// Brief: Master Arm Master Slave Control
FUNCTION_BLOCK PUBLIC FB_StateCtrlInit EXTENDS FB_MasterArmCtrlBase
VAR_INPUT
END_VAR
VAR_OUTPUT
END_VAR
VAR
	m_jnt7SelfCheckVel : LREAL :=180*g_deg2Rad;
	m_jnt7HalfMotionRange : LREAL := 1.75*PI+0.26;
	m_jnt7LimitErr :LREAL := 5*g_deg2Rad;
	m_jnt7CenterPos :LREAL;
	// 0: driver on; 1: joint 7 move to upper limit, 2: joint 7 mvoe to center
	m_initState :INT :=0;
END_VAR

// override this function in each exact controller
METHOD PROTECTED calcCmdJntPos : BOOL

VAR_IN_OUT CONSTANT
	i_slaveIdx :INT;
	i_shoulderPose :ST_Frame;
	i_masterArm :FB_MasterArm;
	i_slaveStatus :ST_SlaveStatus;
END_VAR

VAR
	centerVel:LREAL;
//	curJntPos:Vec7d;
END_VAR
IF m_isFinished THEN
	RETURN;
END_IF

IF m_timePeriod > 1 THEN
	m_isFinished :=true;
END_IF
//CASE m_initState OF
//	0:
//		m_cmdJntPos := i_masterArm.curJntPos;
//		IF i_masterArm.isEnabled(m_jntEnableFlag) = TRUE THEN
//			m_initState :=1;
//		END_IF
//	1: 
//		m_cmdJntPos[7] := m_cmdJntPos[7] + m_jnt7SelfCheckVel * g_armCtrlCycleTime;
//		IF m_cmdJntPos[7]-i_masterArm.curJntPos[7] > m_jnt7LimitErr THEN
//			m_cmdJntPos[7]:=i_masterArm.curJntPos[7];
//			m_jnt7CenterPos :=m_cmdJntPos[7]-m_jnt7HalfMotionRange;
//			m_initState :=2;
//		END_IF
//	2:
//		centerVel :=LIMIT(-m_jnt7SelfCheckVel,(m_jnt7CenterPos-m_cmdJntPos[7])/g_armCtrlCycleTime,m_jnt7SelfCheckVel);
//		m_cmdJntPos[7] := m_cmdJntPos[7] + centerVel * g_armCtrlCycleTime;
//		IF ABS(m_jnt7CenterPos-i_masterArm.curJntPos[7]) < g_jntCtrlAngTolLow THEN
//			m_isFinished :=TRUE;
//		END_IF
//END_CASE
END_METHOD

METHOD PUBLIC init : BOOL
VAR_IN_OUT CONSTANT
	i_masterArm	:FB_MasterArm;
END_VAR
VAR_IN_OUT 
	r_masterArmCtrlCmd :ST_ArmCtrlCmds;
END_VAR

VAR
	i:INT;
END_VAR
SUPER^.Init(i_masterArm,r_masterArmCtrlCmd);
m_jntOPMode:=g_allPosMode;
m_initState :=0;

m_jntOPMode := g_allPosTrqMode;
END_METHOD

END_FUNCTION_BLOCK

(* stored: Version 1.1.0.1, ProductVersion 3.1.4024.12
   POU FB_StateCtrlInit: Id {2f1b91d8-ebd5-4b63-92d8-450fe3a94973}, SpecialFunc None
   Method calcCmdJntPos: Id {b37c9272-afc7-4cb0-8e50-360f85145053}
   Method init: Id {0eca198b-2030-4cc0-a250-a6bdc9d0e230} *)
